TYPE I16 : INT; END_TYPE

(* stored: Version 1.1.0.1
   DUT I16: Id {f64cc5b4-f4fd-067e-2751-a18b9b14ec42} *)
